// TIA Portal project "AventicsEMV" (V19)

(* hardware
DEVICE "S7-1200-Station_1"  S7-1200 Station
   slot 0: "Baugruppenträger_0"  S7-1200 Rack  Rack  V1.0
   slot 1: "PLC_1"  CPU 1215C DC/DC/DC  6ES7 215-1AG40-0XB0  V4.2
   slot 2: "SM 1278_1"  4SI IO link  6ES7 278-4BD32-0XB0  V2.1
DEVICE "HMI_1"  KTP400 Basic PN
   slot 0: "HMI_1"  KTP400 Basic PN  6AV2 123-2DB03-0AX0  15.1.0.0
   slot 1: "HMI_RT_1"  KTP400 Basic PN  6AV2 123-2DB03-0AX0  15.1.0.0
   slot 5: "HMI_1.IE_CP_1"  PROFINET Interface  15.0.1.0
      slot 1: "PROFINET Schnittstelle_1"  PROFINET Interface
         slot 1: "Port_1"  Port
*)

// ===== PLC "PLC_1"  CPU 1215C DC/DC/DC =====

VAR_GLOBAL   // PLC tag table "Standard-Variablentabelle"
   "value" AT %IW69 : Word;
   "ProzessDaten" AT %I8.0 : "PII - NSE-S3 138 IOL";
END_VAR

VAR_GLOBAL   // PLC tag table "Hardware"
   "AnalogInUp" AT %IW64 : Word;
   "AnalogInDown" AT %IW66 : Word;
   "HWIA" AT %I0.0 : "InputsA";
   "HWIB" AT %I1.0 : "InputsB";
   "HWOA" AT %Q0.0 : "OutputsA";
   "HWOB" AT %Q1.0 : "OutputsB";
END_VAR

TYPE "InputsA"
   STRUCT
      INPUTA : Array[0..7] of Bool;
   END_STRUCT;
END_TYPE

TYPE "OutputsA"
   STRUCT
      OUTPUTA : Array[0..7] of Bool;
   END_STRUCT;
END_TYPE

TYPE "InputsB"
   STRUCT
      INPUTB : Array[0..5] of Bool;
   END_STRUCT;
END_TYPE

TYPE "OutputsB"
   STRUCT
      OUTPUTB : Array[0..1] of Bool;
   END_STRUCT;
END_TYPE

TYPE "ICID_1"
   STRUCT
      StatusBytes : Array[0..3] of Byte;
      SampleCounter : Byte;
   END_STRUCT;
END_TYPE

TYPE "ICID_2"
   STRUCT
      Temperatur : Real;
      Force_Torque : Array[0..7] of Real;
   END_STRUCT;
END_TYPE

TYPE "BytesToRead"
   STRUCT
      ByteSet : Array[0..7] of Byte;
   END_STRUCT;
END_TYPE

TYPE "DataSequence"
   STRUCT
      Seq : Array[0..254, 0..3] of UInt;
   END_STRUCT;
END_TYPE

TYPE "ICOD"
   STRUCT
      CommandWord : Byte;
      SelectToolSetting : Byte;
      SelectNoiseReductionFilter : Byte;
   END_STRUCT;
END_TYPE

TYPE "RegisterSequence"
   STRUCT
      RegSequence : Array[0..254, 0..2] of UInt;
   END_STRUCT;
END_TYPE

TYPE "ErrorSequence"
   STRUCT
      ErrorBufferSeq : Array[0..200, 0..6] of UInt;
      Commands : Array[0..200, 0..1] of Bool;
   END_STRUCT;
END_TYPE

TYPE "PII - NSE-S3 138 IOL"
   STRUCT
      "PD Input - Gerätestatus - Bit 0: Betriebsbereit" : Bool;
      "PD Input - Gerätestatus - Bit 1: Warnung" : Bool;
      "PD Input - Gerätestatus - Bit 2: Fehler" : Bool;
      "Reserved Bit" : Bool;
      "Reserved Bit_1" : Bool;
      "Reserved Bit_2" : Bool;
      "PD Input - Gerätestatus - Bit 6: Teachvorgang läuft" : Bool;
      "Reserved Bit_3" : Bool;
      "PD Input - Spannzustand -Bit 0: Gespannt mit Palette" : Bool;
      "PD Input - Spannzustand - Bit 1: Geöffnet" : Bool;
      "PD Input - Spannzustand - Bit 2: Gespannt" : Bool;
      "PD Input - Spannzustand - Bit 3: Geschlossen ohne Bolzen" : Bool;
      "Reserved Bit_4" : Bool;
      "Reserved Bit_5" : Bool;
      "PD Input - Spannzustand - Bit 6: Turbodruck an" : Bool;
      "PD Input - Spannzustand - Bit 7: Palette erkannt" : Bool;
      "Reserved Byte" : Bool;
      "PD Input - Gerätetemperatur" : Byte;
      "PD Input - Anwesenheitssensor (Reserviert 1)" : Real;
      "PD Input - Spannschiebersensor (Reserviert 2)" : Real;
      "PD Input - Drucksensor (Reserviert 3)" : Real;
   END_STRUCT;
END_TYPE

DATA_BLOCK "VariablenM"   // DB1
{ S7_Optimized_Access := 'TRUE' }
VERSION : 0.1
   VAR
      ResetValues : Bool;
      minDruck : Real;
      maxDruck : Real;
      minSpann : Real;
      maxSpann : Real;
      minAws : Real;
      maxAws : Real;
      BolzenState : Byte := 16#01;
      DelayTrigger : Bool;
      ET_Time : Time;
      TimeOutTrigger : Bool;
      oldState : Byte;
      ToggleBit : Bool;
      Start : Bool;
   END_VAR
BEGIN
END_DATA_BLOCK

// folder: ReadWriteFunctins

DATA_BLOCK "WriteFunction_DB"   // DB2
{ S7_Optimized_Access := 'TRUE' }
VERSION : 0.1
// stored: InstanceOfName WriteFunction
"WriteFunction"
BEGIN
END_DATA_BLOCK

DATA_BLOCK "ReadFunction_DB"   // DB6
{ S7_Optimized_Access := 'TRUE' }
VERSION : 0.1
// stored: InstanceOfName ReadFunction
"ReadFunction"
BEGIN
END_DATA_BLOCK

// folder: System blocks/Program resources

DATA_BLOCK "Delay"   // DB4
{ S7_Optimized_Access := 'TRUE' }
AUTHOR : Simatic
FAMILY : IEC
NAME : IEC_TMR
VERSION : 1.0
// stored: InstanceOfName IEC_TIMER
"IEC_TIMER"
BEGIN
END_DATA_BLOCK

DATA_BLOCK "TimeOUT"   // DB8
{ S7_Optimized_Access := 'TRUE' }
AUTHOR : Simatic
FAMILY : IEC
NAME : IEC_TMR
VERSION : 1.0
// stored: InstanceOfName IEC_TIMER
"IEC_TIMER"
BEGIN
END_DATA_BLOCK

// folder: (top level)

FUNCTION "SchaltRoutine" : Void   // FC1, FBD
{ S7_Optimized_Access := 'TRUE' }
VERSION : 0.1
   VAR_TEMP
      Trigger : Bool;
      i : Byte;
   END_VAR
BEGIN

REGION Network 1: Geschlossen ohne Bolzen mit TurboDruck-AN
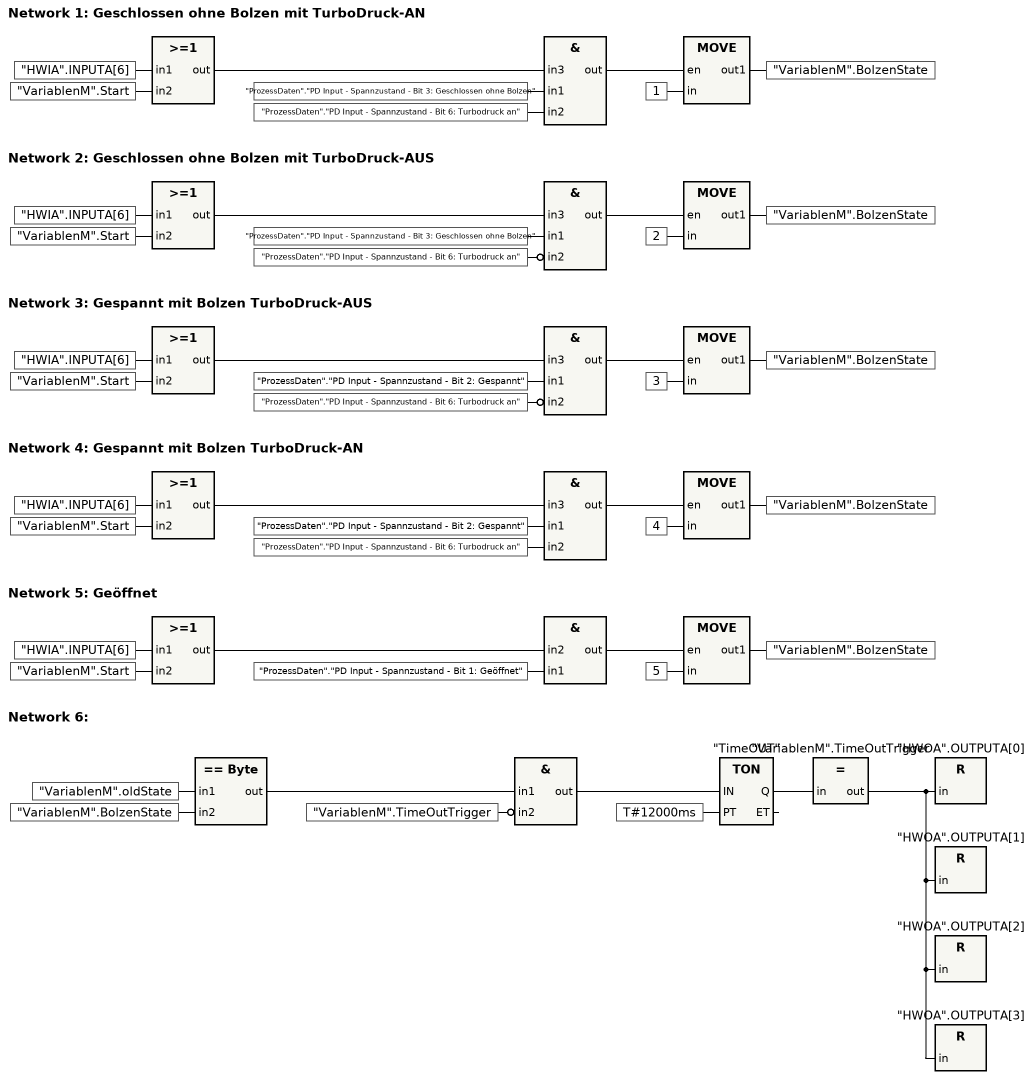
   IF ("HWIA".INPUTA[6] OR "VariablenM".Start) AND "ProzessDaten"."PD Input - Spannzustand - Bit 3: Geschlossen ohne Bolzen" AND "ProzessDaten"."PD Input - Spannzustand - Bit 6: Turbodruck an" THEN
       "VariablenM".BolzenState := 1;
   END_IF;
END_REGION

REGION Network 2: Geschlossen ohne Bolzen mit TurboDruck-AUS
   IF ("HWIA".INPUTA[6] OR "VariablenM".Start) AND "ProzessDaten"."PD Input - Spannzustand - Bit 3: Geschlossen ohne Bolzen" AND NOT "ProzessDaten"."PD Input - Spannzustand - Bit 6: Turbodruck an" THEN
       "VariablenM".BolzenState := 2;
   END_IF;
END_REGION

REGION Network 3: Gespannt mit Bolzen TurboDruck-AUS
   IF ("HWIA".INPUTA[6] OR "VariablenM".Start) AND "ProzessDaten"."PD Input - Spannzustand - Bit 2: Gespannt" AND NOT "ProzessDaten"."PD Input - Spannzustand - Bit 6: Turbodruck an" THEN
       "VariablenM".BolzenState := 3;
   END_IF;
END_REGION

REGION Network 4: Gespannt mit Bolzen TurboDruck-AN
   IF ("HWIA".INPUTA[6] OR "VariablenM".Start) AND "ProzessDaten"."PD Input - Spannzustand - Bit 2: Gespannt" AND "ProzessDaten"."PD Input - Spannzustand - Bit 6: Turbodruck an" THEN
       "VariablenM".BolzenState := 4;
   END_IF;
END_REGION

REGION Network 5: Geöffnet
   IF ("HWIA".INPUTA[6] OR "VariablenM".Start) AND "ProzessDaten"."PD Input - Spannzustand - Bit 1: Geöffnet" THEN
       "VariablenM".BolzenState := 5;
   END_IF;
END_REGION

REGION Network 6
   "TimeOUT".TON(IN := ("VariablenM".oldState = "VariablenM".BolzenState) AND NOT "VariablenM".TimeOutTrigger,
                 PT := T#12000ms);
   "VariablenM".TimeOutTrigger := "TimeOUT".Q;
   IF "TimeOUT".Q THEN
       "HWOA".OUTPUTA[0] := FALSE;
       "HWOA".OUTPUTA[1] := FALSE;
       "HWOA".OUTPUTA[2] := FALSE;
       "HWOA".OUTPUTA[3] := FALSE;
   END_IF;
END_REGION

REGION Network 7 (SCL)
   "Delay".TON(IN:="VariablenM".DelayTrigger,
               PT:=T#5000ms);

   "VariablenM".ET_Time := "Delay".ET;
   "VariablenM".DelayTrigger := TRUE;

   IF "Delay".Q AND ("HWIA".INPUTA[6] OR "VariablenM".Start) THEN
       CASE "VariablenM".BolzenState OF
           1:  // Geschlossen ohne Bolzen TurboDruck-AN
               "HWOA".OUTPUTA[3] := FALSE;
               "HWOA".OUTPUTA[1] := FALSE;
           2:  // Geschlossen ohne Bolzen TurboDruck-Aus
               IF "VariablenM".oldState = 1 OR "VariablenM".oldState = 2 THEN
                   "HWOA".OUTPUTA[2] := TRUE;
                   "HWOA".OUTPUTA[0] := TRUE;
               ELSE
                   "HWOA".OUTPUTA[1] := TRUE;
                   "HWOA".OUTPUTA[3] := TRUE;
               END_IF;
           3:  // Gespannt mit Bolzen TurboDruck-Aus
               IF "VariablenM".oldState = 4 OR "VariablenM".oldState = 3 THEN
                   "HWOA".OUTPUTA[2] := TRUE;
                   "HWOA".OUTPUTA[0] := TRUE;
               ELSE
                   "HWOA".OUTPUTA[3] := TRUE;
                   "HWOA".OUTPUTA[1] := TRUE;
               END_IF;
           4:  // Gespannt mit Bolzen TurboDruck-An
               "HWOA".OUTPUTA[3] := FALSE;
               "HWOA".OUTPUTA[1] := FALSE;
           5:  //Geöffnet
               "HWOA".OUTPUTA[2] := FALSE;
               "HWOA".OUTPUTA[0] := FALSE;
           ELSE  // Statement section ELSE
               ;
       END_CASE;
       "VariablenM".oldState := "VariablenM".BolzenState;
       "VariablenM".DelayTrigger := FALSE;
   END_IF;
END_REGION
END_FUNCTION

FUNCTION "MinMax" : Void   // FC2, SCL
{ S7_Optimized_Access := 'TRUE' }
VERSION : 0.1
BEGIN
   IF "VariablenM".ResetValues THEN
       "VariablenM".minDruck := "ProzessDaten"."PD Input - Drucksensor (Reserviert 3)";
       "VariablenM".maxDruck := "ProzessDaten"."PD Input - Drucksensor (Reserviert 3)";
       "VariablenM".minAws := "ProzessDaten"."PD Input - Anwesenheitssensor (Reserviert 1)";
       "VariablenM".maxAws := "ProzessDaten"."PD Input - Anwesenheitssensor (Reserviert 1)";
       "VariablenM".maxSpann := "ProzessDaten"."PD Input - Spannschiebersensor (Reserviert 2)";
       "VariablenM".minSpann := "ProzessDaten"."PD Input - Spannschiebersensor (Reserviert 2)";
   END_IF;


   IF NOT ("VariablenM".ResetValues) THEN
       IF "VariablenM".minDruck > "ProzessDaten"."PD Input - Drucksensor (Reserviert 3)" THEN
           "VariablenM".minDruck := "ProzessDaten"."PD Input - Drucksensor (Reserviert 3)";
       END_IF;
       IF "VariablenM".maxDruck < "ProzessDaten"."PD Input - Drucksensor (Reserviert 3)" THEN
           "VariablenM".maxDruck := "ProzessDaten"."PD Input - Drucksensor (Reserviert 3)";
       END_IF;

       IF "VariablenM".minSpann > "ProzessDaten"."PD Input - Spannschiebersensor (Reserviert 2)" THEN
           "VariablenM".minSpann := "ProzessDaten"."PD Input - Spannschiebersensor (Reserviert 2)";
       END_IF;
       IF "VariablenM".maxSpann < "ProzessDaten"."PD Input - Spannschiebersensor (Reserviert 2)" THEN
           "VariablenM".maxSpann := "ProzessDaten"."PD Input - Spannschiebersensor (Reserviert 2)";
       END_IF;

       IF "VariablenM".minAws > "ProzessDaten"."PD Input - Anwesenheitssensor (Reserviert 1)" THEN
           "VariablenM".minAws := "ProzessDaten"."PD Input - Anwesenheitssensor (Reserviert 1)";
       END_IF;
       IF "VariablenM".maxAws < "ProzessDaten"."PD Input - Anwesenheitssensor (Reserviert 1)" THEN
           "VariablenM".maxAws := "ProzessDaten"."PD Input - Anwesenheitssensor (Reserviert 1)";
       END_IF;
   END_IF;
END_FUNCTION

ORGANIZATION_BLOCK "Main"   // OB1, FBD, ProgramCycle
TITLE = "Main Program Sweep (Cycle)"
{ S7_Optimized_Access := 'TRUE' }
VERSION : 0.1
   VAR_INPUT
      Initial_Call : Bool;   // Initial call of this OB
      Remanence : Bool;   // =True, if remanent data are available
   END_VAR
   VAR_TEMP
      TempStr : String;
   END_VAR
BEGIN

REGION Network 1
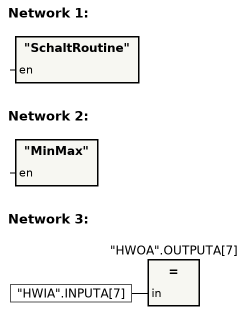
   "SchaltRoutine"();
END_REGION

REGION Network 2
   "MinMax"();
END_REGION

REGION Network 3
   "HWOA".OUTPUTA[7] := "HWIA".INPUTA[7];
END_REGION
END_ORGANIZATION_BLOCK

ORGANIZATION_BLOCK "CLKInterrupt"   // OB30, FBD, CyclicInterrupt
{ S7_Optimized_Access := 'TRUE' }
VERSION : 0.1
   VAR_INPUT
      Initial_Call : Bool;   // Initial call of this OB
      Event_Count : Int;   // Events discarded
   END_VAR
BEGIN

REGION Network 1 (SCL)
   "VariablenM".ToggleBit := NOT ("VariablenM".ToggleBit);
END_REGION
END_ORGANIZATION_BLOCK

// folder: RandomGenerator

FUNCTION_BLOCK "NmbrGenerator"   // FB4, SCL
{ S7_Optimized_Access := 'TRUE' }
VERSION : 0.1
   VAR_INPUT
      min : UInt;
      valueInput : UInt;
      max : UInt;
   END_VAR
   VAR_OUTPUT
      randomNumber : UInt;
   END_VAR
   VAR
      zyklusCNT : UInt;
   END_VAR
   VAR_TEMP
      range : UInt;
   END_VAR
BEGIN
   #zyklusCNT := #zyklusCNT + #valueInput;

   IF #zyklusCNT > 10000 THEN
       #zyklusCNT := 0;
   END_IF;

   // Pseudo-Zufallszahl innerhalb des Bereichs min bis max berechnen
   #range := #max - #min +1;
   IF #range > 0 THEN
       // Pseudo-Zufallszahl durch Modulo-Berechnung
       #randomNumber := #min + (#zyklusCNT MOD #range);
   END_IF;
END_FUNCTION_BLOCK

// folder: ReadWriteFunctins

FUNCTION_BLOCK "WriteFunction"   // FB1, FBD
{ S7_Optimized_Access := 'TRUE' }
VERSION : 0.1
   VAR RETAIN
      ByteToSend : Byte := 16#01;
   END_VAR
   VAR
      Bytes : Byte;
      data : Array[0..3] of Byte;
   END_VAR
   VAR_TEMP
      reqReady : Bool;
   END_VAR
   VAR CONSTANT
      frqIndex : DInt := 16#4020;
      index : DInt := 16#4020;
   END_VAR
   // data[0] := 16#03;
BEGIN

REGION Network 1
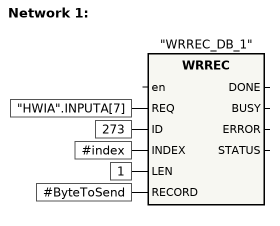
   "WRREC_DB_1"(REQ := "HWIA".INPUTA[7], ID := 273, INDEX := #index, LEN := 1, RECORD := #ByteToSend);   // WRREC
END_REGION
END_FUNCTION_BLOCK

FUNCTION_BLOCK "ReadFunction"   // FB2, FBD
{ S7_Optimized_Access := 'TRUE' }
VERSION : 0.1
   VAR RETAIN
      ByteToSend : Byte := 16#01;
   END_VAR
   VAR CONSTANT
      index : DInt := 16#4020;
   END_VAR
BEGIN

REGION Network 1
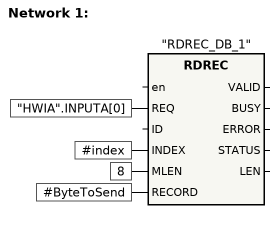
   "RDREC_DB_1"(REQ := "HWIA".INPUTA[0], INDEX := #index, MLEN := 8, RECORD := #ByteToSend);   // RDREC
END_REGION
END_FUNCTION_BLOCK

// ===== library types =====

TYPE "PaketStruct"
   STRUCT
      "+" : Byte;
      "-" : Byte;
      Led : Bool;
      Nummer : Byte;
      Operand : Bool;
   END_STRUCT;
END_TYPE

(* ===== HMI "HMI_RT_1" =====

ScreenModuleEditorView "Bildbaustein_1" 640x480
   Button "Schaltfläche_1" at 176,96 size 96x32; TextOff 'Text'
*)

(* ===== HMI "HMI_RT_1" =====
system functions are stored by id; their names below are inferred from use
connection "HMI_Verbindung_1": ETHERNET, SMART_S7_1200_OMS

HMI tags "Standard-Variablentabelle"
   "HWOA" : OutputsA = PLC HWOA AT %Q0.0, 1 s
   "ProzessDaten" : PII - NSE-S3 138 IOL = PLC ProzessDaten AT %I8.0, 1 s
   "Start" : Bool = PLC VariablenM.Start, 1 s
   "minDruck" : Real = PLC VariablenM.minDruck AT %DB1.DBX0.0, 1 s
   "maxDruck" : Real = PLC VariablenM.maxDruck AT %DB1.DBD0, 1 s
   "minSpann" : Real = PLC VariablenM.minSpann AT %DB1.DBD0, 1 s
   "maxSpann" : Real = PLC VariablenM.maxSpann AT %DB1.DBD0, 1 s
   "minAws" : Real = PLC VariablenM.minAws AT %DB1.DBD0, 1 s
   "maxAws" : Real = PLC VariablenM.maxAws AT %DB1.DBD0, 1 s
   "Reset" : Bool = PLC VariablenM.ResetValues AT %DB1.DBX0.0, 1 s

text list "Textliste_Bildnamen": 1 'Grundbild'

Template "Vorlage_2" 480x272
   GraphicView "Vorlage_Grafikanzeige_1" at -10,0 size 490x277; Picture "Grafik_3"
   Softkey "Softkey_F1" at 0,0 size 0x0
      on KeyDown: ActivateScreen("Bild_1", 0)
   Softkey "Softkey_F2" at 0,0 size 0x0
      on KeyDown: ActivateScreen("Kurve", 0)

screen "Bild_1" 480x272, template "Vorlage_2"
   IOField "EA-Feld_1" at 357,55 size 96x32; FormatPattern 9999.99
      ProcessValue <- "PD Input - Anwesenheitssensor (Reserviert 1)"
   Button "Schaltfläche_1" at 223,9 size 112x253; TextOff 'Stop'
      on Click: ActivateScreen("Bild_2", 0); ResetBit("Start")
   TextField "Textfeld_1" at 385,22 size 39x23; Text 'Aws'
   IOField "EA-Feld_2" at 357,130 size 96x32; FormatPattern 9999.99
      ProcessValue <- "PD Input - Spannschiebersensor (Reserviert 2)"
   TextField "Textfeld_2" at 343,97 size 123x23; Text 'Spannschieber'
   IOField "EA-Feld_3" at 357,205 size 96x32; FormatPattern 9999.99
      ProcessValue <- "PD Input - Drucksensor (Reserviert 3)"
   TextField "Textfeld_3" at 352,172 size 105x23; Text 'Drucksensor'
   TextField "Textfeld_4" at 13,16 size 97x42; Text 'Gespannt mit Palette'
   TextField "Textfeld_5" at 13,64 size 76x23; Text 'Geöffnet'
   TextField "Textfeld_6" at 13,94 size 82x23; Text 'Gespannt'
   TextField "Textfeld_7" at 13,123 size 105x42; Text 'Geschlossen ohne Bolzen'
   TextField "Textfeld_8" at 13,172 size 98x23; Text 'Turbodruck'
   TextField "Textfeld_9" at 13,202 size 69x42; Text 'Palette erkannt'
   Rectangle "Rechteck_1" at 131,27 size 78x21
      Appearance <- "PD Input - Spannzustand -Bit 0: Gespannt mit Palette"
   Rectangle "Rechteck_2" at 131,68 size 78x16
      Appearance <- "PD Input - Spannzustand - Bit 1: Geöffnet"
   Rectangle "Rechteck_3" at 131,98 size 78x16
      Appearance <- "PD Input - Spannzustand - Bit 2: Gespannt"
   Rectangle "Rechteck_4" at 131,133 size 78x23
      Appearance <- "PD Input - Spannzustand - Bit 3: Geschlossen ohne Bolzen"
   Rectangle "Rechteck_5" at 131,176 size 78x16
      Appearance <- "PD Input - Spannzustand - Bit 6: Turbodruck an"
   Rectangle "Rechteck_6" at 131,211 size 79x24
      Appearance <- "PD Input - Spannzustand - Bit 7: Palette erkannt"

screen "Bild_2" 480x272, template "Vorlage_2"
   IOField "EA-Feld_1" at 357,55 size 96x32; FormatPattern 9999.99
      ProcessValue <- "PD Input - Anwesenheitssensor (Reserviert 1)"
   Button "Schaltfläche_1" at 223,9 size 112x253; TextOff 'Start'
      on Click: SetBit("Start"); ActivateScreen("Bild_1", 0)
   TextField "Textfeld_1" at 385,22 size 39x23; Text 'Aws'
   IOField "EA-Feld_2" at 357,130 size 96x32; FormatPattern 9999.99
      ProcessValue <- "PD Input - Spannschiebersensor (Reserviert 2)"
   TextField "Textfeld_2" at 343,97 size 123x23; Text 'Spannschieber'
   IOField "EA-Feld_3" at 357,205 size 96x32; FormatPattern 9999.99
      ProcessValue <- "PD Input - Drucksensor (Reserviert 3)"
   TextField "Textfeld_3" at 352,172 size 105x23; Text 'Drucksensor'
   TextField "Textfeld_4" at 13,16 size 97x42; Text 'Gespannt mit Palette'
   TextField "Textfeld_5" at 13,64 size 76x23; Text 'Geöffnet'
   TextField "Textfeld_6" at 13,94 size 82x23; Text 'Gespannt'
   TextField "Textfeld_7" at 13,123 size 105x42; Text 'Geschlossen ohne Bolzen'
   TextField "Textfeld_8" at 13,172 size 98x23; Text 'Turbodruck'
   TextField "Textfeld_9" at 13,202 size 69x42; Text 'Palette erkannt'
   Rectangle "Rechteck_1" at 131,27 size 78x21
      Appearance <- "PD Input - Spannzustand -Bit 0: Gespannt mit Palette"
   Rectangle "Rechteck_2" at 131,68 size 78x16
      Appearance <- "PD Input - Spannzustand - Bit 1: Geöffnet"
   Rectangle "Rechteck_3" at 131,98 size 78x16
      Appearance <- "PD Input - Spannzustand - Bit 2: Gespannt"
   Rectangle "Rechteck_4" at 131,133 size 78x23
      Appearance <- "PD Input - Spannzustand - Bit 3: Geschlossen ohne Bolzen"
   Rectangle "Rechteck_5" at 131,176 size 78x16
      Appearance <- "PD Input - Spannzustand - Bit 6: Turbodruck an"
   Rectangle "Rechteck_6" at 131,211 size 79x24
      Appearance <- "PD Input - Spannzustand - Bit 7: Palette erkannt"

screen "Kurve" 480x272, template "Vorlage_2"
   IOField "EA-Feld_7" at 101,55 size 98x48; FormatPattern 9999.99
      ProcessValue <- "minAws"
   TextField "Textfeld_7" at 37,63 size 39x23; Text 'Aws'
   TextField "Textfeld_8" at 19,115 size 73x42; Text 'Spann- schieber'
   TextField "Textfeld_9" at 25,177 size 59x42; Text 'Druck- sensor'
   TextField "Textfeld_1" at 133,25 size 96x23; Text 'Min'
   TextField "Textfeld_2" at 365,25 size 96x23; Text 'Max'
   TextField "Textfeld_3" at 247,26 size 96x23; Text 'Live'
   IOField "EA-Feld_1" at 101,116 size 98x48; FormatPattern 9999.99
      ProcessValue <- "minSpann"
   IOField "EA-Feld_2" at 101,177 size 98x48; FormatPattern 9999.99
      ProcessValue <- "minDruck"
   IOField "EA-Feld_3" at 217,55 size 98x48; FormatPattern 9999.99
      ProcessValue <- "PD Input - Anwesenheitssensor (Reserviert 1)"
   IOField "EA-Feld_4" at 217,116 size 98x48; FormatPattern 9999.99
      ProcessValue <- "PD Input - Spannschiebersensor (Reserviert 2)"
   IOField "EA-Feld_5" at 217,177 size 98x48; FormatPattern 9999.99
      ProcessValue <- "PD Input - Drucksensor (Reserviert 3)"
   IOField "EA-Feld_6" at 337,55 size 98x48; FormatPattern 9999.99
      ProcessValue <- "maxAws"
   IOField "EA-Feld_8" at 337,116 size 98x48; FormatPattern 9999.99
      ProcessValue <- "maxSpann"
   IOField "EA-Feld_9" at 337,177 size 98x48; FormatPattern 9999.99
      ProcessValue <- "maxDruck"
   Button "Schaltfläche_1" at 11,9 size 80x54; TextOff 'Reset'
      on Press: SetBit("Reset")
      on Release: ResetBit("Reset")
*)